{attribute 'qualified_only'}
VAR_GLOBAL
	bStartButton: BOOL;
	bStopButton: BOOL;
	fVelocity: REAL;
	fAccelleration: REAL;
	
	//Output
	nMotorPosition: LREAL;
	bMotorEnabled: BOOL;
	bMotorForward: BOOL;
	bMotorBackwards: BOOL;
	
	//Internal
	axis: AXIS_REF;
	fBJog: MC_Jog;
	fBPower: MC_Power;
END_VAR

(* stored: Version 1.1.0.1, ProductVersion 3.1.4024.12
   GVL GVL: Id {bb0c83e5-da50-46c2-b200-b3c47f3fa699} *)
